REGION Network 256: Update Job History
   // Update the History of jobs if a new job was started
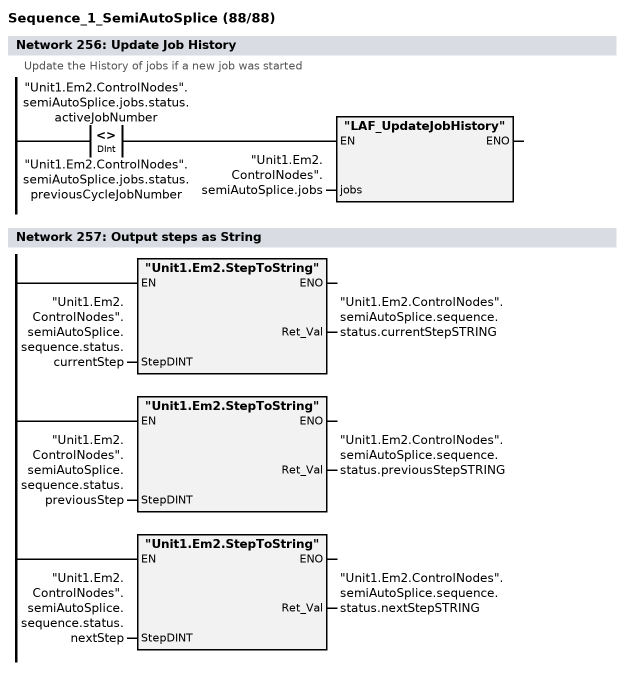
   RUNG wire#powerrail
      { S7_Templates := "SrcType := DInt" } NE_Contact(in1 := "Unit1.Em2.ControlNodes".semiAutoSplice.jobs.status.activeJobNumber, in2 := "Unit1.Em2.ControlNodes".semiAutoSplice.jobs.status.previousCycleJobNumber)
      "LAF_UpdateJobHistory"(jobs := "Unit1.Em2.ControlNodes".semiAutoSplice.jobs)
   END_RUNG
   // the same network as SCL:
   IF "Unit1.Em2.ControlNodes".semiAutoSplice.jobs.status.activeJobNumber <> "Unit1.Em2.ControlNodes".semiAutoSplice.jobs.status.previousCycleJobNumber THEN
       "LAF_UpdateJobHistory"(jobs := "Unit1.Em2.ControlNodes".semiAutoSplice.jobs);
   END_IF;
END_REGION

REGION Network 257: Output steps as String
   RUNG wire#powerrail
      "Unit1.Em2.StepToString"(StepDINT := "Unit1.Em2.ControlNodes".semiAutoSplice.sequence.status.currentStep, Ret_Val => "Unit1.Em2.ControlNodes".semiAutoSplice.sequence.status.currentStepSTRING)
   END_RUNG
   RUNG wire#powerrail
      "Unit1.Em2.StepToString"(StepDINT := "Unit1.Em2.ControlNodes".semiAutoSplice.sequence.status.previousStep, Ret_Val => "Unit1.Em2.ControlNodes".semiAutoSplice.sequence.status.previousStepSTRING)
   END_RUNG
   RUNG wire#powerrail
      "Unit1.Em2.StepToString"(StepDINT := "Unit1.Em2.ControlNodes".semiAutoSplice.sequence.status.nextStep, Ret_Val => "Unit1.Em2.ControlNodes".semiAutoSplice.sequence.status.nextStepSTRING)
   END_RUNG
   // the same network as SCL:
   "Unit1.Em2.ControlNodes".semiAutoSplice.sequence.status.currentStepSTRING := "Unit1.Em2.StepToString"(StepDINT := "Unit1.Em2.ControlNodes".semiAutoSplice.sequence.status.currentStep);
   "Unit1.Em2.ControlNodes".semiAutoSplice.sequence.status.previousStepSTRING := "Unit1.Em2.StepToString"(StepDINT := "Unit1.Em2.ControlNodes".semiAutoSplice.sequence.status.previousStep);
   "Unit1.Em2.ControlNodes".semiAutoSplice.sequence.status.nextStepSTRING := "Unit1.Em2.StepToString"(StepDINT := "Unit1.Em2.ControlNodes".semiAutoSplice.sequence.status.nextStep);
END_REGION
END_FUNCTION_BLOCK
